FUNCTION_BLOCK ChangeModeOnAllSubModulesVisitor IMPLEMENTS I_ModuleVisitor
VAR
	TargetMode	 : DINT;
	Statemachine : I_ContainStatemachine;
END_VAR

METHOD ChangeMode
VAR_INPUT
	TargetMode : DINT;
	Module	   : I_Module;
END_VAR
THIS^.TargetMode := TargetMode;
Module.Modules.Accept(THIS^);
END_METHOD

METHOD VisitModule
VAR_INPUT
	Module : I_Module;
END_VAR
IF __QUERYINTERFACE(Module, Statemachine) THEN
	Statemachine.Statemachine.Mode.ChangeMode(THIS^.TargetMode);
END_IF
END_METHOD

END_FUNCTION_BLOCK

(* stored: Version 1.1.0.1, ProductVersion 3.1.4026.18
   POU ChangeModeOnAllSubModulesVisitor: Id {06c2fc4a-1392-454e-868a-04379af90dab}, SpecialFunc None
   Method ChangeMode: Id {0690df9b-48d7-4c8f-b3e9-ccacd6e7ded7}
   Method VisitModule: Id {440d1907-7f96-441d-bb6f-0b8b66e4a51d} *)
